(****************************************************************************************)
(*							Beckhoff Automation Poland									*)
(*								F_2ndByteW v1.0											*)
(*									15.02.2010											*)
(*		Funkcja wyciagajaca bardziej znaczacy BYTE ze zmiennej typu WORD				*)
(*							 wyjscie typu WORD											*)
(*______________________________________________________________________________________*)
FUNCTION F_2ndByteW : WORD
VAR_INPUT
	wIn		:	WORD;
END_VAR

F_2ndByteW := wIn AND 16#FF00;

END_FUNCTION

(* stored: Version 1.1.0.1, ProductVersion 3.1.4020.3
   POU F_2ndByteW: Id {d7729598-0167-4e2e-97d8-772dce6237b9}, SpecialFunc None *)
